// TIA Portal V20 export
// export: Created 2026-10-03T18:54:34.3833094Z, ExportSetting WithDefaults, DisplayName Totally Integrated Automation Portal, DisplayVersion V20 Update 4, DisplayName TIA Portal Openness, DisplayVersion V20 Update 4, DisplayName TIA Portal Version Control Interface, DisplayVersion V20 Update 4, DisplayName SINAMICS Startdrive Advanced, DisplayVersion V20 SP1 Update 1, DisplayName SINAMICS Startdrive G110M, G120, G120C, G120D, G120P, G115D, DisplayVersion V20 SP1 Update 1, DisplayName SINAMICS Startdrive G130, G150, S120, S150, SINAMICS MV, G220, S200, S210, DisplayVersion V20 SP1 Update 1, DisplayName STEP 7 Professional, DisplayVersion V20 Update 4, DisplayName STEP 7 Safety, DisplayVersion V20 Update 2, DisplayName WinCC Basic/Comfort/Advanced, DisplayVersion V20 Update 4, DisplayName WinCC Unified, DisplayVersion V20 Update 4
FUNCTION "SLC_WORD_WRITE" : Void   // FC15, SCL
TITLE = Write a whole word of a bit file
{ S7_Optimized_Access := 'TRUE' }
VERSION : 0.1
// Writes B<File>:<Element> as a number, for SLC logic that wrote a whole word of a bit file (MOV N7:100 B3:16,
//  CLR B3:5, ...). All 16 named bits of that word change together, as in the SLC.
// stored: AutoNumber true, IsIECCheckEnabled false, SetENOAutomatically false, UDAEnableTagReadback false
   VAR_INPUT
      File : DInt;   // Bit file number (3 for B3)
      Element : DInt;   // Word number (16 for B3:16)
      Value : Int;   // New value of the word
   END_VAR
BEGIN
   // 16#84 is the DB memory area; each word is 2 bytes.
   POKE(area := 16#84, dbNumber := #File, byteOffset := #Element * 2, value := INT_TO_WORD(#Value));
END_FUNCTION
